KUKA KRL data list: CADMATCH_BASIC.dat

&ACCESS RVP
&REL 1
&PARAM EDITMASK = *
DEFDAT CADMATCH_BASIC
ENDDAT
